//PowerOn=0
IF Autoflow=0 AND SystemReadyStatus AND NOT(bErrorTHBack) AND NOT(bErrorTHOut) AND AutoStatus  THEN
	Autoflow:=1;
END_IF;

(*Idle=1*)
TON_1(IN:= Autoflow=1 AND NOT(bObjSNR) ,PT:= tNoObjDelayTime);
IF Autoflow=1 AND (bFeedStart) THEN
	Autoflow:=2;
END_IF;
(*無料,節流出=2*)
IF Autoflow=2 THEN
	ObjSNRStatus:=FALSE;
END_IF;

IF Autoflow=2 AND bTHOutLS THEN
	Autoflow:=3;
END_IF;
(*到出,平送起振=3*)
IF Autoflow=3 AND bObjSNR THEN
	ObjSNRStatus:=TRUE;
END_IF;
TON_2(IN:= Autoflow=3 AND bObjSNR ,PT:= tObjectExistDelayTime);
TON_3(IN:= Autoflow=3 AND NOT(bObjSNR) ,PT:= t#4s);
IF TON_3.Q THEN
	bFeedError:=TRUE;
END_IF;
IF bReset THEN
	bFeedError:=FALSE;
END_IF;

IF Autoflow=3 AND TON_2.Q AND NOT(bFeedError) THEN
	Autoflow:=4;
END_IF;
(*工件到位,平送停振=4*)
IF Autoflow=4 THEN
	Autoflow:=5;
END_IF;
(*節流回=5*)
IF Autoflow=5 AND bTHBackLS THEN
	Autoflow:=6;
END_IF;
(*節流到回=6*)
IF Autoflow=6 THEN
	bFeedFinish:=TRUE;
	ELSE
	bFeedFinish:=FALSE;
END_IF;

IF Autoflow=6 AND NOT(bFeedStart) THEN
	Autoflow:=1;
END_IF;
(*************************************************************************)
(*Error*)
R_TRIG_3(CLK:=bErrorTHBack);
R_TRIG_4(CLK:=bErrorTHOut);

IF NOT(SystemReadyStatus) OR NOT(AutoStatus) OR bErrorTHBack OR bErrorTHOut THEN
	Autoflow:=0;
END_IF;

(*************************************************************************)
(*手動*)
(*節流*)
R_TRIG_1(CLK:=bTHPB AND NOT(AutoStatus));
(*SET*)
IF (((R_TRIG_1.Q) AND NOT(THStatus)) OR Autoflow=2 OR R_TRIG_3.Q) AND bInterlock_thout THEN
	bTHSOL:=TRUE;
END_IF;
(*RESET*)
IF (((R_TRIG_1.Q) AND THStatus) OR Autoflow=5 OR R_TRIG_4.Q) AND bInterlock_thback THEN
	bTHSOL:=FALSE;
END_IF;
(*STATE*)
THStatus:=bTHSOL;

(*平送*)
(*輸出*)
bFeedRY:=Autoflow=2 OR Autoflow=3 OR bSupplierRY OR bTHSOL;
END_FUNCTION_BLOCK